FUNCTION_BLOCK TPulseTimer
VAR
    TP1 : TP;
END_VAR

METHOD FB_init : BOOL
VAR_INPUT
	bInitRetains : BOOL; // if TRUE, the retain variables are initialized (warm start / cold start)
	bInCopyCode : BOOL;  // if TRUE, the instance afterwards gets moved into the copy code (online change)
    PresetTime : LREAL; // seconds
END_VAR
TP1.PT := LREAL_TO_TIME(PresetTime * 1000);
END_METHOD

PROPERTY OutputState : BOOL
GET
OutputState := TP1.Q;
END_GET
END_PROPERTY

PROPERTY PresetTime : LREAL
GET
PresetTime := TIME_TO_LREAL(TP1.PT)/1000.0; // in seconds
END_GET
SET
TP1.PT := LREAL_TO_TIME(PresetTime * 1000);
END_SET
END_PROPERTY

METHOD Pulse : BOOL
VAR_INPUT
    In : BOOL;
END_VAR
TP1(IN := In);
Pulse := TP1.Q;
END_METHOD

METHOD Reset
TP1(IN := FALSE);
END_METHOD

METHOD Run : BOOL
TP1(IN := TRUE);
Run := TP1.Q;
END_METHOD

END_FUNCTION_BLOCK

(* stored: Version 1.1.0.1, ProductVersion 3.1.4024.3
   POU TPulseTimer: Id {6f05ebc1-646f-0297-12f6-3bc75caab056}, SpecialFunc None
   Method FB_init: Id {e2b11b30-67e2-050e-0fb0-e3f3555327eb}
   Property OutputState: Id {68059222-9a8a-0581-2f56-efd6a810cf5c}
   Get Get: Id {48f9aa2d-9ec7-02c5-121a-cc89fb8d806b}
   Property PresetTime: Id {471f1ec6-dbcb-0c44-1d09-6f49a42994dd}
   Get Get: Id {e75fc37d-0a84-07d4-35af-998e47490717}
   Set Set: Id {aa4864df-2e13-0fa2-28ac-7b22a5370c7b}
   Method Pulse: Id {f03700c9-6c18-0988-086b-61a9f7e66e11}
   Method Reset: Id {c5405954-40bf-0829-270c-59d5a7f6ec90}
   Method Run: Id {d7881203-1b2d-0d85-0052-70ffb08afca4} *)
